# EPICS autosave request: iocBoot/iocEPU1/motor.req
$(SYS){$(DEV)-$(AXIS)}-Mtr.VELO
$(SYS){$(DEV)-$(AXIS)}-Mtr.ACCL
